// SIMATIC S7-200 SMART project (STEP 7-Micro/WIN SMART), CPU ST40

SYMBOL_TABLE Table 1
Start_SW         I0.0
Stop_SW          I0.1
Timer            T1
Motor_1          Q0.0
Motor_2          Q0.1
END_SYMBOL_TABLE

ORGANIZATION_BLOCK MAIN:OB1
TITLE=Program Comments
BEGIN
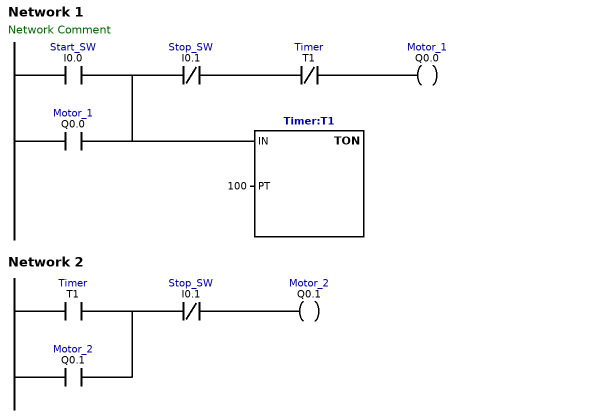
Network 1
// Network Comment
// (network saved uncompiled; LAD cells follow)
// row 0: c0 -| |- Start_SW:I0.0 v  c1 -|/|- Stop_SW:I0.1  c2 -|/|- Timer:T1  c3 -( ) Motor_1:Q0.0
// row 1: c0 -| |- Motor_1:Q0.0 ^  c1 --  c2 [TON Timer:T1 IN:=power@row1, PT:=100]
// row 2: c2 [box]
Network 2
LD     Timer:T1
O      Motor_2:Q0.1
AN     Stop_SW:I0.1
=      Motor_2:Q0.1
END_ORGANIZATION_BLOCK
